{attribute 'GeneratedUsingTerminal: EL1262-0000-0002'}
{attribute addProperty BoxType "EL1262-0000-0002"}
{attribute addProperty Id "DcOutputShiftAT %I*DINT4DcInputShiftAT %I*DINT4StateAT %I*UINT2"}
{attribute addProperty CRC "2806213574"}
{attribute addProperty Size "10"}
TYPE InfoData_A7436BC6 :
STRUCT
	{attribute addProperty Name "DcOutputShift"}
	DcOutputShift AT %I* : DINT;
	{attribute addProperty Name "DcInputShift"}
	DcInputShift AT %I* : DINT;
	{attribute addProperty Name "State"}
	State AT %I* : UINT;
END_STRUCT
END_TYPE

(* stored: Version 1.2.0.0, ProductVersion 3.1.4024.9
   DUT InfoData_A7436BC6: Id {f5098cc2-cb5a-4a16-b82b-add1a413fcef} *)
